PROGRAM P_InkSystem
VAR

END_VAR

P_ISS();
P_Stirrer_WastePump();

END_PROGRAM

(* stored: Version 1.1.0.1, ProductVersion 3.1.4024.11
   POU P_InkSystem: Id {d9a0afbc-418e-46e5-90d4-34e152ff11fa}, SpecialFunc None *)
